// TIA Portal project "s7_1200" (V16)

(* hardware
DEVICE "S7-1200 station_1"  S7-1200 Station
   slot 0: "Rack_0"  S7-1200 Rack  Rack  V1.0
   slot 1: "Quicksilver"  CPU 1211C DC/DC/DC  6ES7 211-1AE40-0XB0  V4.4
*)

// ===== PLC "Quicksilver"  CPU 1211C DC/DC/DC =====

VAR_GLOBAL   // PLC tag table "Default tag table"
   "ledQ0" AT %Q0.0 : Bool;
   "ledQ1" AT %Q0.1 : Bool;
   "ledQ2" AT %Q0.2 : Bool;
   "ain_0" AT %IW64 : Int;   // IW is reading metric, bool for pulse
   "ain_1" AT %IW66 : Int;   // IW is reading metric, bool for pulse
   "aout_0" AT %QD0 : Real;
   "aout_1" AT %QD1 : Real;
   "offset" AT %MW68 : Int;   // Signal 2 - Holds offset for pulse
   "base" AT %MW70 : Int;   // Holds the base value for pulse
   "error" AT %Q0.3 : Bool;   // Error for out-of-range values
   "temp_base" AT %MW72 : Int;   // Temporary base to track changes on base
   "temp_signal1" AT %MW74 : Int;   // Signal 1
   "temp_out" AT %MW76 : Int;
   "System_Byte" AT %MB1 : Byte;
   "FirstScan" AT %M1.0 : Bool;
   "DiagStatusUpdate" AT %M1.1 : Bool;
   "AlwaysTRUE" AT %M1.2 : Bool;
   "AlwaysFALSE" AT %M1.3 : Bool;
   "Clock_Byte" AT %MB0 : Byte;
   "Clock_10Hz" AT %M0.0 : Bool;
   "Clock_5Hz" AT %M0.1 : Bool;
   "Clock_2.5Hz" AT %M0.2 : Bool;
   "Clock_2Hz" AT %M0.3 : Bool;
   "Clock_1.25Hz" AT %M0.4 : Bool;
   "Clock_1Hz" AT %M0.5 : Bool;
   "Clock_0.625Hz" AT %M0.6 : Bool;
   "Clock_0.5Hz" AT %M0.7 : Bool;
END_VAR

DATA_BLOCK "MB_Config"   // DB2
{ S7_Optimized_Access := 'TRUE' }
VERSION : 0.1
   VAR
      DISCONNECT : Bool;
      MB_MODE : USInt := 0;   // MB_MODE=0: Read, MB_MODE=1 and 2: Writing
      DATA_ADDR : UDInt := 40001;   // Start Address: 40001
      DATA_LEN : UDInt;   // Data Length: 10
      CONNECT : TCON_IP_v4;
      DONE : Bool;
      BUSY : Bool;
      ERROR : Bool;
      STATUS : Word;
   END_VAR
BEGIN
   CONNECT.InterfaceId := 64;
   CONNECT.ID := 1;
   CONNECT.ConnectionType := 11;
   CONNECT.ActiveEstablished := true;
   CONNECT.RemoteAddress.ADDR[1] := 10;
   CONNECT.RemoteAddress.ADDR[2] := 83;
   CONNECT.RemoteAddress.ADDR[3] := 64;
   CONNECT.RemoteAddress.ADDR[4] := 70;
   CONNECT.RemotePort := 502;
   // CONNECT.RemoteAddress.ADDR : Address of Server to connect to!
END_DATA_BLOCK

DATA_BLOCK "MB_Buffer"   // DB3
{ S7_Optimized_Access := 'TRUE' }
VERSION : 0.1
   VAR
      DATA : Array[0..9] of Word;
   END_VAR
BEGIN
END_DATA_BLOCK

ORGANIZATION_BLOCK "Main_modbus"   // OB1, LAD, ProgramCycle
TITLE = "Main Program Sweep (Cycle)"
{ S7_Optimized_Access := 'TRUE' }
VERSION : 0.1
   VAR_INPUT
      Initial_Call : Bool;   // Initial call of this OB
      Remanence : Bool;   // =True, if remanent data are available
   END_VAR
BEGIN

REGION Network 1
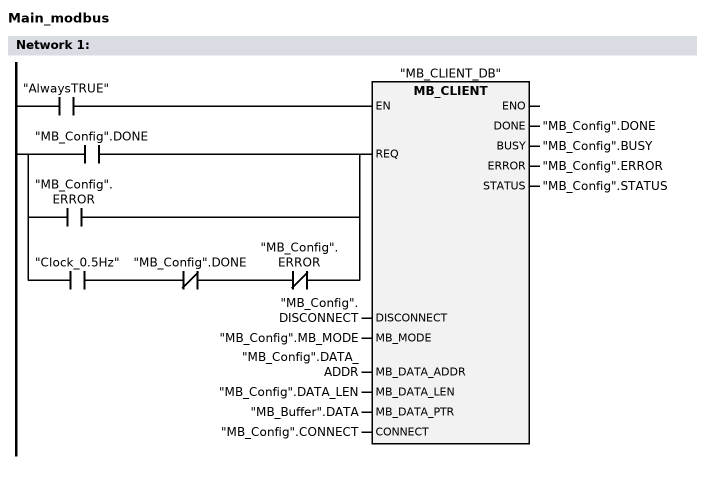
   IF "AlwaysTRUE" THEN
       "MB_CLIENT_DB"(REQ := "MB_Config".DONE OR "MB_Config".ERROR OR ("Clock_0.5Hz" AND NOT "MB_Config".DONE AND NOT "MB_Config".ERROR),   // MB_CLIENT
                      DISCONNECT := "MB_Config".DISCONNECT,
                      MB_MODE := "MB_Config".MB_MODE,
                      MB_DATA_ADDR := "MB_Config".DATA_ADDR,
                      MB_DATA_LEN := "MB_Config".DATA_LEN,
                      MB_DATA_PTR := "MB_Buffer".DATA,
                      CONNECT := "MB_Config".CONNECT,
                      DONE => "MB_Config".DONE,
                      BUSY => "MB_Config".BUSY,
                      ERROR => "MB_Config".ERROR,
                      STATUS => "MB_Config".STATUS);
   END_IF;
END_REGION
END_ORGANIZATION_BLOCK

ORGANIZATION_BLOCK "Double_Pulse"   // OB123, LAD, ProgramCycle
TITLE = "Main Program Sweep (Cycle)"
{ S7_Optimized_Access := 'TRUE' }
VERSION : 0.1
   VAR_INPUT
      Initial_Call : Bool;   // Initial call of this OB
      Remanence : Bool;   // =True, if remanent data are available
   END_VAR
   VAR_TEMP   // added for the SCL form of the ladder/FBD networks
      _w1 : Bool;
      _w2 : Bool;
   END_VAR
BEGIN

REGION Network 1: Receive offset from AIN_1
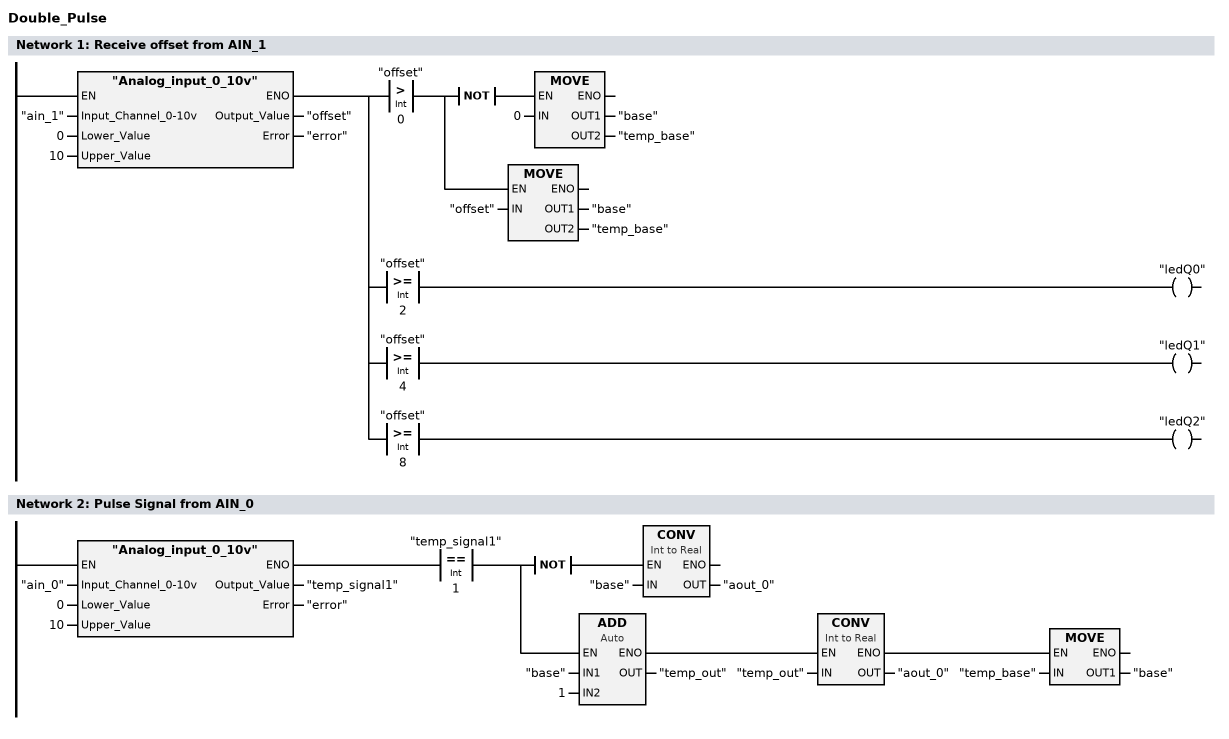
   RUNG wire#powerrail
      "Analog_input_0_10v"("Input_Channel_0-10v" := "ain_1", Lower_Value := 0, Upper_Value := 10, Output_Value => "offset", Error => "error")
      wire#w1
      { S7_Templates := "SrcType := Int" } GT_Contact(in1 := "offset", in2 := 0)
      wire#w2
      Not()
      Move(in := 0, out1 => "base", out2 => "temp_base")
   END_RUNG
   RUNG wire#w2
      Move(in := "offset", out1 => "base", out2 => "temp_base")
   END_RUNG
   RUNG wire#w1
      { S7_Templates := "SrcType := Int" } GE_Contact(in1 := "offset", in2 := 2)
      Coil( "ledQ0" )
   END_RUNG
   RUNG wire#w1
      { S7_Templates := "SrcType := Int" } GE_Contact(in1 := "offset", in2 := 4)
      Coil( "ledQ1" )
   END_RUNG
   RUNG wire#w1
      { S7_Templates := "SrcType := Int" } GE_Contact(in1 := "offset", in2 := 8)
      Coil( "ledQ2" )
   END_RUNG
   // the same network as SCL:
   "Analog_input_0_10v"("Input_Channel_0-10v" := "ain_1",
                        Lower_Value := 0,
                        Upper_Value := 10,
                        Output_Value => "offset",
                        Error => "error",
                        ENO => #_w1);
   #_w2 := #_w1 AND ("offset" > 0);
   IF NOT #_w2 THEN
       "base" := 0;
       "temp_base" := 0;
   END_IF;
   IF #_w2 THEN
       "base" := "offset";
       "temp_base" := "offset";
   END_IF;
   "ledQ0" := #_w1 AND ("offset" >= 2);
   "ledQ1" := #_w1 AND ("offset" >= 4);
   "ledQ2" := #_w1 AND ("offset" >= 8);
END_REGION

REGION Network 2: Pulse Signal from AIN_0
   RUNG wire#powerrail
      "Analog_input_0_10v"("Input_Channel_0-10v" := "ain_0", Lower_Value := 0, Upper_Value := 10, Output_Value => "temp_signal1", Error => "error")
      { S7_Templates := "SrcType := Int" } EQ_Contact(in1 := "temp_signal1", in2 := 1)
      wire#w1
      Not()
      { S7_Templates := "[SrcType := Int, DestType := Real]" } Convert(in := "base", out => "aout_0")
   END_RUNG
   RUNG wire#w1
      Add(in1 := "base", in2 := 1, out => "temp_out")
      { S7_Templates := "[SrcType := Int, DestType := Real]" } Convert(in := "temp_out", out => "aout_0")
      Move(in := "temp_base", out1 => "base")
   END_RUNG
   // the same network as SCL:
   "Analog_input_0_10v"("Input_Channel_0-10v" := "ain_0",
                        Lower_Value := 0,
                        Upper_Value := 10,
                        Output_Value => "temp_signal1",
                        Error => "error",
                        ENO => #_w1);
   #_w2 := #_w1 AND ("temp_signal1" = 1);
   IF NOT #_w2 THEN "aout_0" := INT_TO_REAL("base"); END_IF;
   IF #_w2 THEN
       "temp_out" := "base" + 1;
       "aout_0" := INT_TO_REAL("temp_out");
       "base" := "temp_base";
   END_IF;
END_REGION
END_ORGANIZATION_BLOCK

// folder: System blocks/Program resources

FUNCTION "Analog_input_0_10v" : Void   // FC1, LAD
{ S7_Optimized_Access := 'TRUE' }
VERSION : 0.1
   VAR_INPUT
      "Input_Channel_0-10v" : Int;
      Lower_Value : Int;
      Upper_Value : Int;
   END_VAR
   VAR_OUTPUT
      Output_Value : Real;
      Error : Bool;
   END_VAR
   VAR_TEMP
      Temp1 : Real;
   END_VAR
BEGIN

REGION Network 1: Bounds check
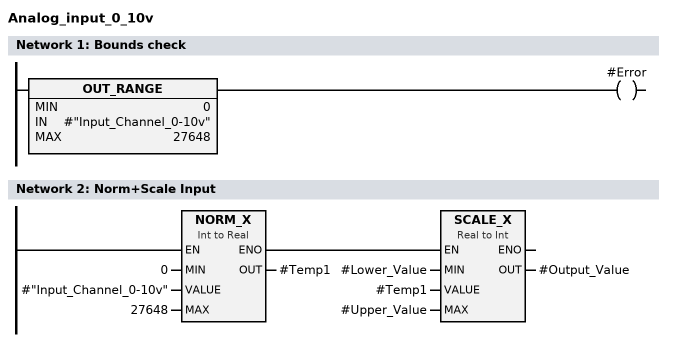
   #Error := (#"Input_Channel_0-10v" < 0) OR (#"Input_Channel_0-10v" > 27648);
END_REGION

REGION Network 2: Norm+Scale Input
   RUNG wire#powerrail
      { S7_Templates := "[SrcType := Int, DestType := Real]" } Normalize(min := 0, value := #"Input_Channel_0-10v", max := 27648, out => #Temp1)
      { S7_Templates := "[SrcType := Real, DestType := Int]" } Scale(min := #Lower_Value, value := #Temp1, max := #Upper_Value, out => #Output_Value)
   END_RUNG
   // the same network as SCL:
   #Temp1 := NORM_X(MIN := 0, VALUE := #"Input_Channel_0-10v", MAX := 27648);
   #Output_Value := SCALE_X(MIN := #Lower_Value, VALUE := #Temp1, MAX := #Upper_Value);
END_REGION
END_FUNCTION